// TIA Portal project "CAA_Lab_Project" (V15)

(* hardware
DEVICE "S71500/ET200MP station_1"  S7-1500 station
   slot 0: "Rail_0"  Rack  6ES7 590-1***0-0AA0
   slot 1: "PLC_1"  CPU 1512C-1 PN  6ES7 512-1CK01-0AB0  V2.5
      slot 3: "CPU display_1"  6ES7591-1AA00-0AA0
DEVICE "HMI_1"  KTP700 Basic PN
   slot 0: "HMI_1"  KTP700 Basic PN  6AV2 123-2GB03-0AX0  15.0.0.0
   slot 1: "HMI_RT_1"  KTP700 Basic PN  6AV2 123-2GB03-0AX0  15.0.0.0
   slot 5: "HMI_1.IE_CP_1"  PROFINET Interface  15.0.0.0
      slot 1: "PROFINET Interface_1"  PROFINET Interface
         slot 1: "Port_1"  Port
*)

// ===== PLC "PLC_1"  CPU 1512C-1 PN =====

VAR_GLOBAL   // PLC tag table "Default tag table"
   "HsePwr" AT %MD0 : Real;
   "FacPwr" AT %MD1 : Real;
   "IndPwr" AT %MD2 : Real;
   "SubLim" AT %MD3 : Real;
   "FacMRun" AT %M4.0 : Bool;
   "CurHr" AT %MW5 : Int;
   "HseTv" AT %M6.0 : Bool;
   "FacLg2" AT %M7.0 : Bool;
   "HseFan" AT %M8.0 : Bool;
   "Mot1" AT %M9.0 : Bool;
   "Mot2" AT %M10.0 : Bool;
   "Mot3" AT %M11.0 : Bool;
   "PkHr" AT %M12.0 : Bool;
   "ShedP3" AT %M16.0 : Bool;
   "ShedP2" AT %M17.0 : Bool;
   "TotPwr" AT %MD18 : Real;
   "ActLim" AT %MD19 : Real;
   "SafeLm" AT %MD20 : Real;
END_VAR

DATA_BLOCK "Substation"   // DB1
{ S7_Optimized_Access := 'TRUE' }
VERSION : 0.1
   VAR RETAIN
      HsePwr : Real := 0.0;
      FacPwr : Real := 0.0;
      IndPwr : Real := 0.0;
      SubLim : Real := 2500.0;
      FacMRun : Bool;
      CurHr : Int := 9;
      HseTvOFF : Bool;
      FacLgON : Bool;
      HseFanOFF : Bool;
      Mot1 : Bool;
      Mot2 : Bool;
      Mot3 : Bool;
      PkHr : Bool;
      ShedP3 : Bool;
      ShedP2 : Bool;
      TotPwr : Real := 0.0;
      SafeLm1 : Real := 0.0;
      SafeLm2 : Real := 0.0;
      HseTVON : Bool := false;
      HseFanoN : Bool := false;
      IndON : Bool;
      HseHL : Bool;
      Warning : Bool;
      FacLgOFF : Bool;
      Mot2OFF : Bool;
      IndHL : Bool;
      "Major Warning" : Bool;
      Danger : Bool;
   END_VAR
BEGIN
END_DATA_BLOCK

// folder: System blocks/Program resources

DATA_BLOCK "IEC_Timer_0_DB"   // DB2
{ S7_Optimized_Access := 'TRUE' }
AUTHOR : Simatic
FAMILY : IEC
NAME : IEC_TMR
VERSION : 1.0
// stored: InstanceOfName IEC_TIMER
"IEC_TIMER"
BEGIN
END_DATA_BLOCK

DATA_BLOCK "TmrM2"   // DB3
{ S7_Optimized_Access := 'TRUE' }
AUTHOR : Simatic
FAMILY : IEC
NAME : IEC_TMR
VERSION : 1.0
// stored: InstanceOfName IEC_TIMER
"IEC_TIMER"
BEGIN
END_DATA_BLOCK

DATA_BLOCK "TmrM3"   // DB4
{ S7_Optimized_Access := 'TRUE' }
AUTHOR : Simatic
FAMILY : IEC
NAME : IEC_TMR
VERSION : 1.0
// stored: InstanceOfName IEC_TIMER
"IEC_TIMER"
BEGIN
END_DATA_BLOCK

// folder: (top level)

ORGANIZATION_BLOCK "Main"   // OB1, LAD, ProgramCycle
TITLE = "Main Program Sweep (Cycle)"
{ S7_Optimized_Access := 'TRUE' }
VERSION : 0.1
   VAR_INPUT
      Initial_Call : Bool;   // Initial call of this OB
      Remanence : Bool;   // =True, if remanent data are available
   END_VAR
BEGIN

REGION Network 1
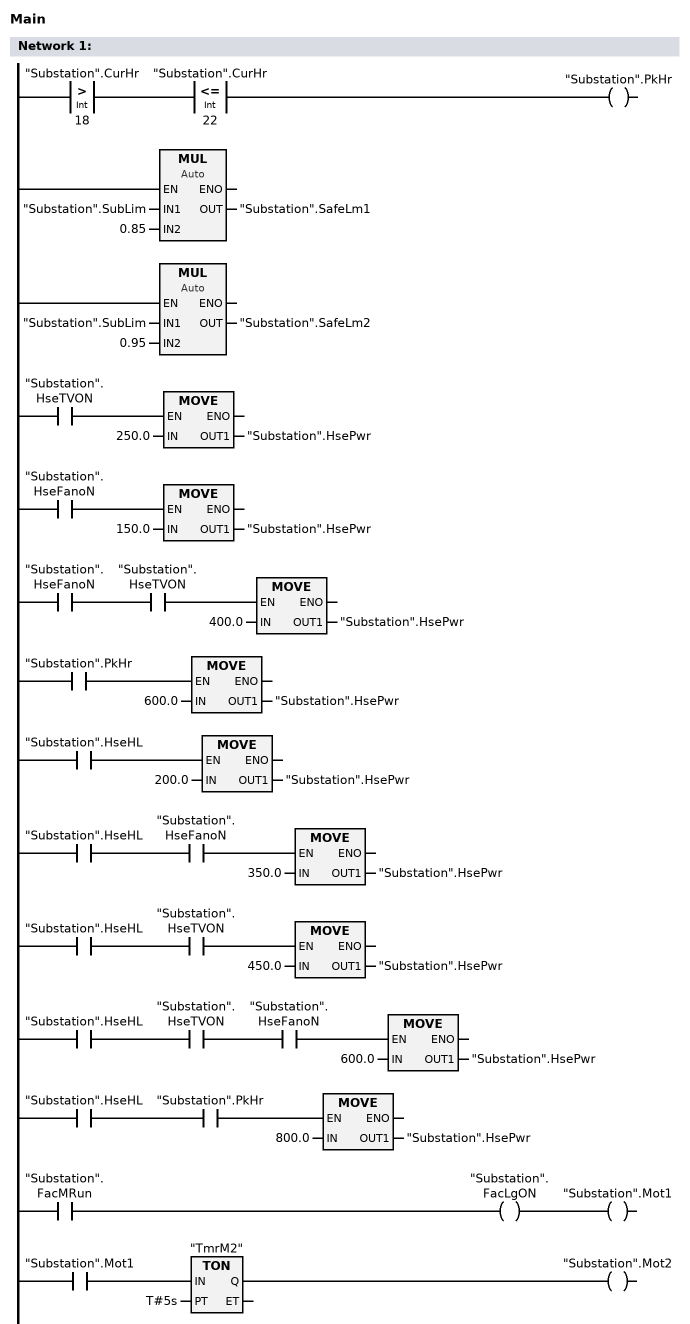
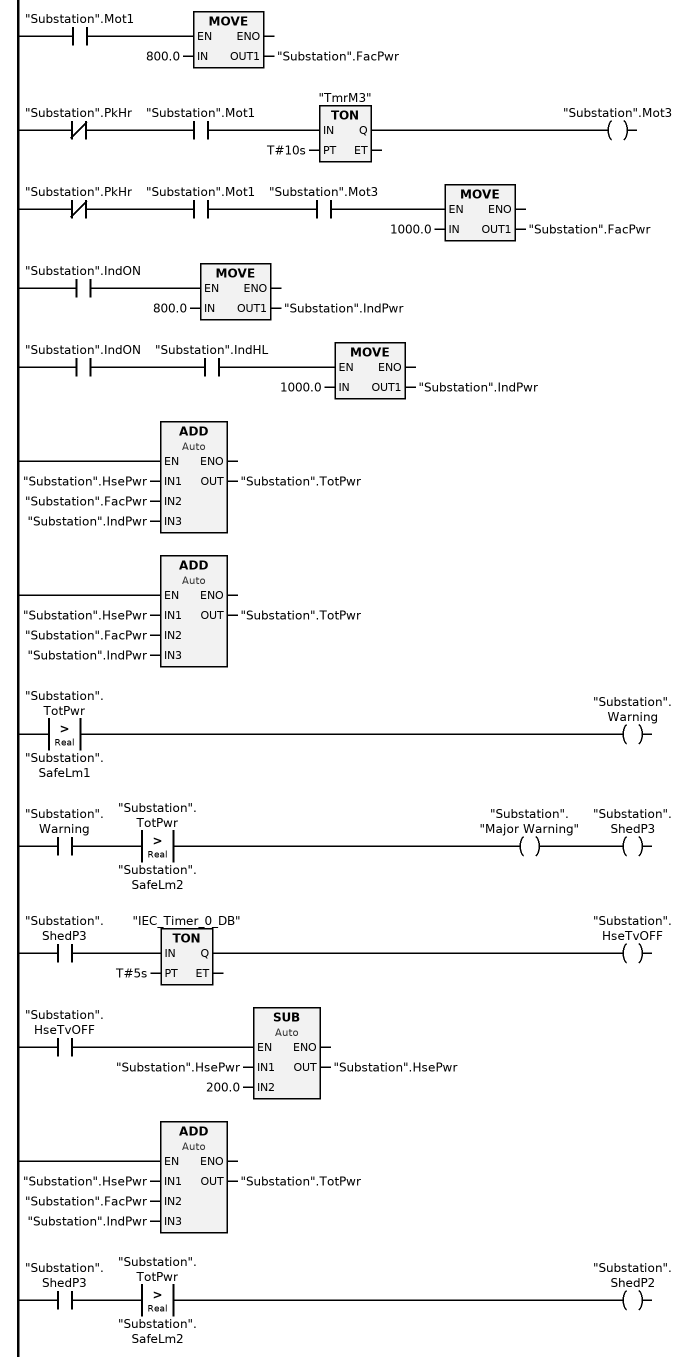
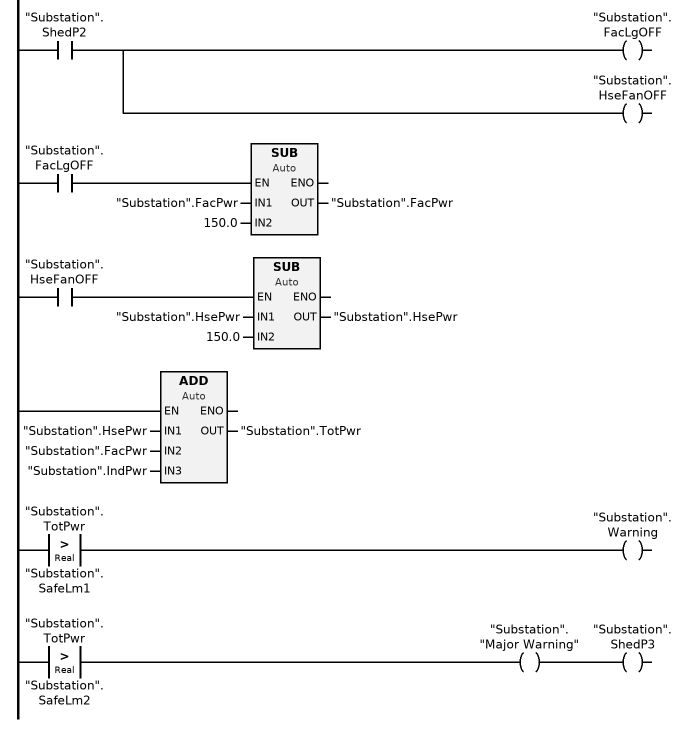
   "Substation".PkHr := ("Substation".CurHr > 18) AND ("Substation".CurHr <= 22);
   "Substation".SafeLm1 := "Substation".SubLim * 0.85;
   "Substation".SafeLm2 := "Substation".SubLim * 0.95;
   IF "Substation".HseTVON THEN "Substation".HsePwr := 250.0; END_IF;
   IF "Substation".HseFanoN THEN "Substation".HsePwr := 150.0; END_IF;
   IF "Substation".HseFanoN AND "Substation".HseTVON THEN "Substation".HsePwr := 400.0; END_IF;
   IF "Substation".PkHr THEN "Substation".HsePwr := 600.0; END_IF;
   IF "Substation".HseHL THEN "Substation".HsePwr := 200.0; END_IF;
   IF "Substation".HseHL AND "Substation".HseFanoN THEN "Substation".HsePwr := 350.0; END_IF;
   IF "Substation".HseHL AND "Substation".HseTVON THEN "Substation".HsePwr := 450.0; END_IF;
   IF "Substation".HseHL AND "Substation".HseTVON AND "Substation".HseFanoN THEN
       "Substation".HsePwr := 600.0;
   END_IF;
   IF "Substation".HseHL AND "Substation".PkHr THEN "Substation".HsePwr := 800.0; END_IF;
   "Substation".FacLgON := "Substation".FacMRun;
   "Substation".Mot1 := "Substation".FacMRun;
   "TmrM2".TON(IN := "Substation".Mot1, PT := T#5s);
   "Substation".Mot2 := "TmrM2".Q;
   IF "Substation".Mot1 THEN "Substation".FacPwr := 800.0; END_IF;
   "TmrM3".TON(IN := NOT "Substation".PkHr AND "Substation".Mot1, PT := T#10s);
   "Substation".Mot3 := "TmrM3".Q;
   IF NOT "Substation".PkHr AND "Substation".Mot1 AND "Substation".Mot3 THEN
       "Substation".FacPwr := 1000.0;
   END_IF;
   IF "Substation".IndON THEN "Substation".IndPwr := 800.0; END_IF;
   IF "Substation".IndON AND "Substation".IndHL THEN "Substation".IndPwr := 1000.0; END_IF;
   "Substation".TotPwr := "Substation".HsePwr + "Substation".FacPwr + "Substation".IndPwr;
   "Substation".TotPwr := "Substation".HsePwr + "Substation".FacPwr + "Substation".IndPwr;
   "Substation".Warning := "Substation".TotPwr > "Substation".SafeLm1;
   "Substation"."Major Warning" := "Substation".Warning AND ("Substation".TotPwr > "Substation".SafeLm2);
   "Substation".ShedP3 := "Substation"."Major Warning";
   "IEC_Timer_0_DB".TON(IN := "Substation".ShedP3, PT := T#5s);
   "Substation".HseTvOFF := "IEC_Timer_0_DB".Q;
   IF "Substation".HseTvOFF THEN "Substation".HsePwr := "Substation".HsePwr - 200.0; END_IF;
   "Substation".TotPwr := "Substation".HsePwr + "Substation".FacPwr + "Substation".IndPwr;
   "Substation".ShedP2 := "Substation".ShedP3 AND ("Substation".TotPwr > "Substation".SafeLm2);
   "Substation".FacLgOFF := "Substation".ShedP2;
   "Substation".HseFanOFF := "Substation".ShedP2;
   IF "Substation".FacLgOFF THEN "Substation".FacPwr := "Substation".FacPwr - 150.0; END_IF;
   IF "Substation".HseFanOFF THEN "Substation".HsePwr := "Substation".HsePwr - 150.0; END_IF;
   "Substation".TotPwr := "Substation".HsePwr + "Substation".FacPwr + "Substation".IndPwr;
   "Substation".Warning := "Substation".TotPwr > "Substation".SafeLm1;
   "Substation"."Major Warning" := "Substation".TotPwr > "Substation".SafeLm2;
   "Substation".ShedP3 := "Substation"."Major Warning";
END_REGION
END_ORGANIZATION_BLOCK

(* ===== HMI "HMI_RT_1" =====
system functions are stored by id; their names below are inferred from use
connection "HMI_Connection_1": ETHERNET, SMART_S7_1500_OMS
connection "HMI_Connection_2": ETHERNET, SMART_S7_1500_OMS

HMI tags "Default tag table"
   "Substation_TotPwr" : Real = PLC Substation.TotPwr, 1 s
   "Substation_HseTVON" : Bool = PLC Substation.HseTVON, 1 s
   "Substation_HseTvOFF" : Bool = PLC Substation.HseTvOFF, 1 s
   "Substation_HsePwr" : Real = PLC Substation.HsePwr, 1 s
   "Substation_HseFanoN" : Bool = PLC Substation.HseFanoN, 1 s
   "Substation_HseHL" : Bool = PLC Substation.HseHL, 1 s
   "Substation_FacMRun" : Bool = PLC Substation.FacMRun, 1 s
   "Substation_FacPwr" : Real = PLC Substation.FacPwr, 1 s
   "Substation_IndON" : Bool = PLC Substation.IndON, 1 s
   "Substation_IndHL" : Bool = PLC Substation.IndHL, 1 s
   "Substation_IndPwr" : Real = PLC Substation.IndPwr, 1 s
   "Substation_CurHr" : Int = PLC Substation.CurHr, 1 s
   "Substation_Warning" : Bool = PLC Substation.Warning, 1 s
   "Substation_Major Warning" : Bool = PLC Substation."Major Warning", 1 s

Template "Template_1" 800x480
   Button "Exit" at 714,429 size 71x50; TextOff 'Exit'; PictureOff "ExitRuntime_KTP700_Basic_PN_TR"; PictureOn "ExitRuntime_KTP700_Basic_PN_TR"
      on Release: StopRuntime(0)
   Button "Template_Button" at 614,429 size 71x50; TextOff 'Text'
   Button "Template_Button_1" at 514,429 size 71x50; TextOff 'Text'
   Button "Template_Button_2" at 414,429 size 71x50; TextOff 'Text'
   Button "Template_Button_3" at 314,429 size 71x50; TextOff 'Text'
   Button "Template_Button_4" at 214,429 size 71x50; TextOff 'Text'
   Button "Template_Button_5" at 114,429 size 71x50; TextOff 'Text'
   Button "Start screen" at 14,429 size 71x50; TextOff 'Start screen'; PictureOff "NavigateHome_KTP700_Basic_PN_TR"; PictureOn "NavigateHome_KTP700_Basic_PN_TR"
      on Release: ActivateScreen("Root screen", 0)

screen "Root screen" 800x480, template "Template_1"
   TextField "HmiScreenItemData" at 80,200 size 640x25; Text 'Text'
   IOField "I/O field_1" at 671,168 size 96x32; FormatPattern 9999999
      ProcessValue <- "Substation_TotPwr"
   TextField "Text field_1" at 662,141 size 105x23; Text 'Total Power'
   Button "Button_1" at 19,43 size 96x32; TextOff 'TV'; TextOn 'TV ON'
      on Click: InvertBit("Substation_HseTVON")
   Button "Button_2" at 21,90 size 96x32; TextOff 'Fan'
      on Click: InvertBit("Substation_HseFanoN")
   Button "Button_3" at 19,143 size 96x32; TextOff 'Grinder'
      on Click: InvertBit("Substation_HseHL")
   TextField "Text field_2" at 44,12 size 52x23; Text 'Home'
   IOField "I/O field_2" at 25,224 size 96x32; FormatPattern 999999999.999
      ProcessValue <- "Substation_HsePwr"
   TextField "Text field_3" at 19,192 size 112x23; Text 'House Power'
   Button "Button_4" at 229,43 size 96x32; TextOff 'Motor ON'
      on Click: InvertBit("Substation_FacMRun")
   IOField "I/O field_3" at 235,128 size 96x32; FormatPattern 999999999.999
      ProcessValue <- "Substation_FacPwr"
   TextField "Text field_4" at 222,99 size 122x23; Text 'Factory Power'
   Button "Button_5" at 410,36 size 96x32; TextOff 'Machine'
      on Click: InvertBit("Substation_IndON")
   TextField "Text field_5" at 235,11 size 69x23; Text 'Factory'
   TextField "Text field_6" at 429,11 size 133x23; Text 'Industry'
   Button "Button_6" at 411,90 size 96x32; TextOff 'Heavy Load'
      on Click: InvertBit("Substation_IndHL")
   IOField "I/O field_4" at 410,160 size 96x32; FormatPattern 999999999.999
      ProcessValue <- "Substation_IndPwr"
   TextField "Text field_7" at 394,133 size 130x23; Text 'Industry Power'
   IOField "I/O field_5" at 662,62 size 96x32; FormatPattern 99999
      ProcessValue <- "Substation_CurHr"
   TextField "Text field_8" at 658,36 size 111x23; Text 'Current Hour'
   Circle "Circle_1" at 429,324 size 48x48
      Appearance <- "Substation_Warning"
   TextField "Text field_9" at 393,375 size 99x23; Text 'Heavy Load'
*)